Universal Robots PolyScope program: CircleWelding.urp

Program CircleWelding (createdIn=3.3.1.237 lastSavedIn=3.3.2.266 directory=/programs/cslnewfolder installation=default robotSerialNumber=2015330057)
Calibrated DH parameters: a=[-0.000017, -0.239459, -0.182322, 0.000061, 0.000089, 0]; d=[0.151941, 5.438834, 44.076234, -49.402704, 0.085399, 0.082167]; alpha=[1.571747, -0.008827, -0.002243, 1.571398, -1.569364, 0]; deltaTheta=[-0.000041, -0.197925, -0.349334, 0.547115, 0.000045, -0.000031]
BeforeStart
  i_Center := Center_feature
  Script: i_Center[3]=0
  Script: i_Center[4]=0
  Script: i_Center[5]=0
Robot Program (runOnlyOnce=false motionType=MoveJ speed=1.047198 acceleration=1.396263 recalculateMotions=false)
  MoveJ speed 60 deg/s, acceleration 80 deg/s^2 (recalculateMotions=false)
    Waypoint HomeWaypoint: TCP in base x=-64.063 y=-289.171 z=12.396 mm, rx=0.5674 ry=2.9848 rz=-0.3523 rad; joints [-74.59, -128.622, -145.021, 17.539, 88.048, 36.914] deg; flange x=-45.005 y=-263.412 z=69.827 mm, rx=0.5675 ry=2.9847 rz=-0.3524 rad
  MoveL speed 250 mm/s, acceleration 1200 mm/s^2 (recalculateMotions=false) feature=Base
    Waypoint FirstWaypoint: TCP in base x=-64.052 y=-284.524 z=-46.768 mm, rx=0.5674 ry=2.9847 rz=-0.3524 rad; joints [-74.241, -151.55, -140.67, 36.113, 87.935, 37.094] deg; flange x=-45.005 y=-258.752 z=10.658 mm, rx=0.5675 ry=2.9847 rz=-0.3524 rad
  var_FirstPose := FirstWaypoint
  pose_Base2Cen := pose_inv(i_Center)
  Pose_Tcp2VarCen := pose_trans(pose_Base2Cen,var_FirstPose)
  Script file /programs/cslnewfolder/CircleWeldingMove.script
    | global DeltaX=var_FirstPose[0]-i_Center[0]
    | global DeltaY=var_FirstPose[1]-i_Center[1]
    | global Weld_Radius=sqrt(DeltaX*DeltaX+DeltaY*DeltaY)
    | global var_Theta_Res=i_Resolution/Weld_Radius
    | global move_count=0
    | global Theta_Delta=0.0
    | global pose_temp1=p[0.0,0.0,0.0,0.0,0.0,0.0]
    | global pose_temp2=p[0.0,0.0,0.0,0.0,0.0,0.0]
    | global pose_VarCenter=i_Center
    | global pose_VarTCP=Pose_Tcp2VarCen
    | global step_time=i_Resolution/0.05
    | global lookaheadTime=0.1
    | overheadTheta=var_Theta_Res*lookaheadTime/step_time+6.2831852
    | while Theta_Delta<=6.2831852:
    |  pose_temp2=pose_trans(pose_VarCenter,pose_VarTCP)
    |  JointPose=get_inverse_kin(pose_temp2)
    |  servoj(JointPose,t=step_time)
    |  move_count=move_count+1
    | 
    |  Theta_Delta=var_Theta_Res*move_count
    |  pose_temp1[5]=Theta_Delta
    |  pose_VarCenter=pose_trans(i_Center,pose_temp1)
    |  pose_VarTCP=pose_trans(Pose_Tcp2VarCen,pose_temp1)
    | end
    | while Theta_Delta<=overheadTheta:
    |  pose_temp2=pose_trans(pose_VarCenter,pose_VarTCP)
    |  JointPose=get_inverse_kin(pose_temp2)
    |  servoj(JointPose,t=step_time)
    |  move_count=move_count+1
    | 
    |  Theta_Delta=var_Theta_Res*move_count
    |  pose_temp1[5]=Theta_Delta
    |  pose_VarCenter=pose_trans(i_Center,pose_temp1)
    |  pose_VarTCP=pose_trans(Pose_Tcp2VarCen,pose_temp1)
    | 
    | end
    | 
    | movel(pose_trans(i_Center,Pose_Tcp2VarCen),a=1.2,v=0.25,r=0)
